FUNCTION_BLOCK INTERNAL FB_IdleState IMPLEMENTS I_State
VAR
	pMachine				: POINTER TO FB_Machine; // Points to the state machine (THIS)
	fVSensors				: ARRAY [0..1] OF REAL; 
END_VAR

METHOD PUBLIC Check 
VAR
	fInputVoltage			: REAL;	
END_VAR
fVSensors := THIS^.pMachine^.VSensors;

fInputVoltage := fVSensors[0];

IF (fInputVoltage >= THIS^.pMachine^.LowerBoundV AND fInputVoltage <= THIS^.pMachine^.UpperBoundV) THEN
	THIS^.pMachine^.Message := '[IDLE]The input voltage is within the boundaries.$0A NOW WAITING FOR ACKNOWLEDGEMENT TO ENTER PRE-CHARGE STATE.';
ELSE
	THIS^.pMachine^.Message := '[IDLE] The input voltage is NOT within the boundaries.$0A SYSTEM ENTERS DISCHARGE STATE.';
	THIS^.pMachine^.SetState(THIS^.pMachine^.DischargeState);
END_IF
END_METHOD

PROPERTY PUBLIC Description : STRING
GET
Description := 'IDLE';
END_GET
END_PROPERTY

METHOD PUBLIC FB_init
VAR_INPUT
	bInitRetains 	: BOOL; // if TRUE, the retain variables are initialized (warm start / cold start)
	bInCopyCode 	: BOOL;  // if TRUE, the instance afterwards gets moved into the copy code (online change)
	pMachine		: POINTER TO FB_Machine; // Points to the state machine (THIS)
END_VAR
THIS^.pMachine := pMachine;
END_METHOD

METHOD PUBLIC PressButton
VAR
	fInputVoltage			: REAL; 
END_VAR
fVSensors := THIS^.pMachine^.VSensors;
fInputVoltage := fVSensors[0];

IF (fInputVoltage >= THIS^.pMachine^.LowerBoundV AND fInputVoltage <= THIS^.pMachine^.UpperBoundV) THEN
	THIS^.pMachine^.Message := '[IDLE] Acknowledge button has been pressed. $0A SYSTEM ENTERS PRECHARGE STATE.';
	THIS^.pMachine^.SetState(THIS^.pMachine^.PrechargeState);
	THIS^.StartTimer();
END_IF
END_METHOD

METHOD PUBLIC PressDischarge
THIS^.pMachine^.Message := '[IDLE] Discharge button has been pressed. $0A SYSTEM ENTERS DISCHARGE STATE.';
THIS^.pMachine^.SetState(THIS^.pMachine^.DischargeState);
END_METHOD

METHOD PUBLIC Reset
THIS^.pMachine^.Message := '[IDLE] Reset button has been pressed. $0A SYSTEM ENTERS DISCHARGE STATE.';
THIS^.pMachine^.SetState(THIS^.pMachine^.DischargeState);
END_METHOD

METHOD PUBLIC StartTimer
THIS^.pMachine^.charge_TON.IN := TRUE; // Starts the Timer
END_METHOD

METHOD PUBLIC Stop
THIS^.pMachine^.SetState(THIS^.pMachine^.ErrorState);
END_METHOD

METHOD PUBLIC TimerDone
END_METHOD

END_FUNCTION_BLOCK

(* stored: Version 1.1.0.1, ProductVersion 3.1.4024.12
   POU FB_IdleState: Id {0a22dcc3-3bc6-4d93-9aca-a747ceef61e5}, SpecialFunc None
   Method Check: Id {89bc70d7-56d9-4f8e-a0cb-7e6c3581ccf8}
   Property Description: Id {4da43970-b44e-45d3-a26f-2725e415c36a}
   Get Get: Id {7741009e-cd74-45df-a568-2e1192ccf97c}
   Method FB_init: Id {5a63751c-4592-4ced-9a19-79495be376cc}
   Method PressButton: Id {9cea9d2f-0f0c-4db1-a5b6-a232015beeb8}
   Method PressDischarge: Id {9ca35365-8866-4214-9a30-90082ff5e02a}
   Method Reset: Id {40dd2636-4e7b-4a6d-8829-9d305a0428d3}
   Method StartTimer: Id {91ecf8e2-0e79-4bd3-8d6b-f4591cb6472b}
   Method Stop: Id {e01351bb-71a2-4811-8728-ab7a48a35088}
   Method TimerDone: Id {c58b6810-c7e7-4af7-8e87-4db08a682ad7} *)
